# EPICS autosave request: ipApp/Db/PTC10_tec_in_settings.req
$(P)$(T):$(C):temperature.SCAN
#$(P)$(T):$(C):sensor
$(P)$(T):$(C):current
